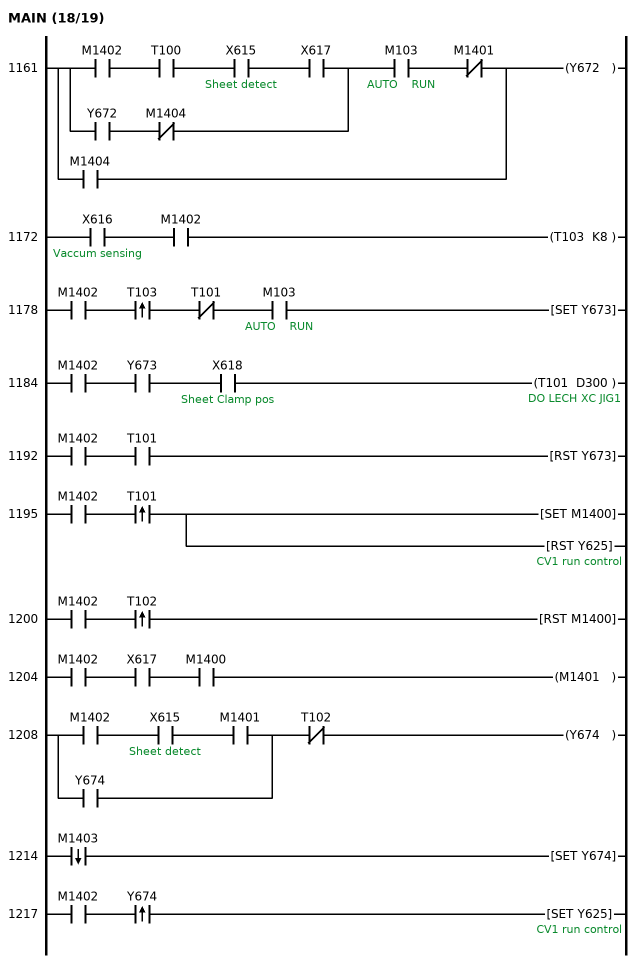
[picture p24: ladder of MAIN, rungs at steps 1161 to 1217]
1161  LD      M1402
      AND     T100
      AND     X615  ; Sheet detect
      AND     X617
      LD      Y672
      ANI     M1404
      ORB
      AND     M103  ; AUTO    RUN
      ANI     M1401
      OR      M1404
      OUT     Y672
1172  LD      X616  ; Vaccum sensing
      AND     M1402
      OUT     T103 K8
1178  LD      M1402
      ANDP    T103
      ANI     T101
      AND     M103  ; AUTO    RUN
      SET     Y673
1184  LD      M1402
      AND     Y673
      AND     X618  ; Sheet Clamp pos
      OUT     T101 D300  ; DO LECH XC JIG1
1192  LD      M1402
      AND     T101
      RST     Y673
1195  LD      M1402
      ANDP    T101
      SET     M1400
      RST     Y625  ; CV1 run control
1200  LD      M1402
      ANDP    T102
      RST     M1400
1204  LD      M1402
      AND     X617
      AND     M1400
      OUT     M1401
1208  LD      M1402
      AND     X615  ; Sheet detect
      AND     M1401
      OR      Y674
      ANI     T102
      OUT     Y674
1214  LDF     M1403
      SET     Y674
1217  LD      M1402
      ANDP    Y674
      SET     Y625  ; CV1 run control
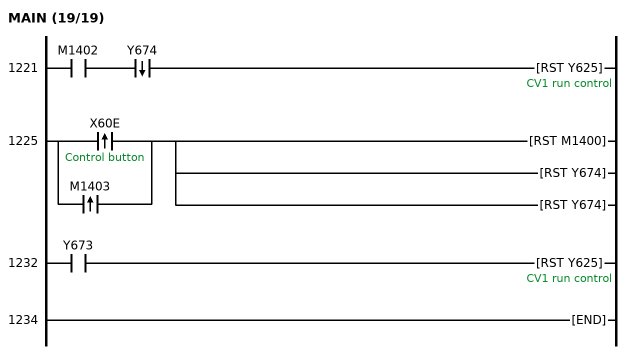
1221  LD      M1402
      ANDF    Y674
      RST     Y625  ; CV1 run control
1225  LDP     X60E  ; Control button
      ORP     M1403
      RST     M1400
      RST     Y674
      RST     Y674
1232  LD      Y673
      RST     Y625  ; CV1 run control
1234  END
END_PROGRAM

PROGRAM MONITOR
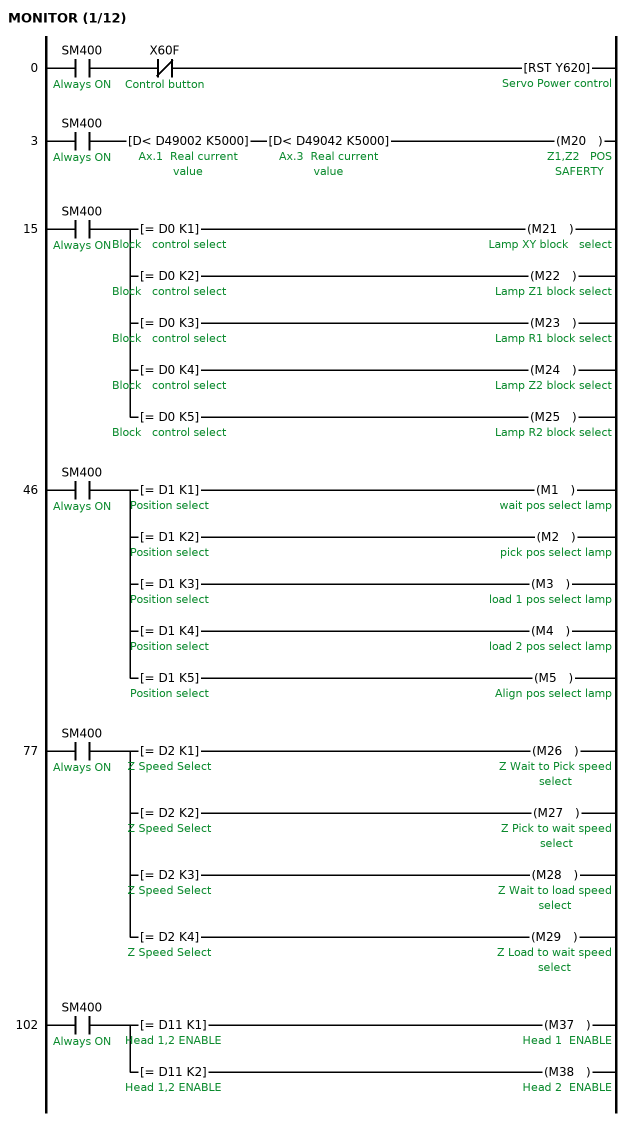
0     LD      SM400  ; Always ON
      ANI     X60F  ; Control button
      RST     Y620  ; Servo Power control
3     LD      SM400  ; Always ON
      ANDD<   D49002 K5000  ; Ax.1  Real current value
      ANDD<   D49042 K5000  ; Ax.3  Real current value
      OUT     M20  ; Z1,Z2   POS     SAFERTY
15    LD      SM400  ; Always ON
      MPS
      AND=    D0 K1  ; Block   control select
      OUT     M21  ; Lamp XY block   select
      MRD
      AND=    D0 K2  ; Block   control select
      OUT     M22  ; Lamp Z1 block select
      MRD
      AND=    D0 K3  ; Block   control select
      OUT     M23  ; Lamp R1 block select
      MRD
      AND=    D0 K4  ; Block   control select
      OUT     M24  ; Lamp Z2 block select
      MPP
      AND=    D0 K5  ; Block   control select
      OUT     M25  ; Lamp R2 block select
46    LD      SM400  ; Always ON
      MPS
      AND=    D1 K1  ; Position select
      OUT     M1  ; wait pos select lamp
      MRD
      AND=    D1 K2  ; Position select
      OUT     M2  ; pick pos select lamp
      MRD
      AND=    D1 K3  ; Position select
      OUT     M3  ; load 1 pos select lamp
      MRD
      AND=    D1 K4  ; Position select
      OUT     M4  ; load 2 pos select lamp
      MPP
      AND=    D1 K5  ; Position select
      OUT     M5  ; Align pos select lamp
77    LD      SM400  ; Always ON
      MPS
      AND=    D2 K1  ; Z Speed Select
      OUT     M26  ; Z Wait to Pick speed select
      MRD
      AND=    D2 K2  ; Z Speed Select
      OUT     M27  ; Z Pick to wait speed select
      MRD
      AND=    D2 K3  ; Z Speed Select
      OUT     M28  ; Z Wait to load speed select
      MPP
      AND=    D2 K4  ; Z Speed Select
      OUT     M29  ; Z Load to wait speed select
102   LD      SM400  ; Always ON
      MPS
      AND=    D11 K1  ; Head 1,2 ENABLE
      OUT     M37  ; Head 1  ENABLE
      MPP
      AND=    D11 K2  ; Head 1,2 ENABLE
      OUT     M38  ; Head 2  ENABLE
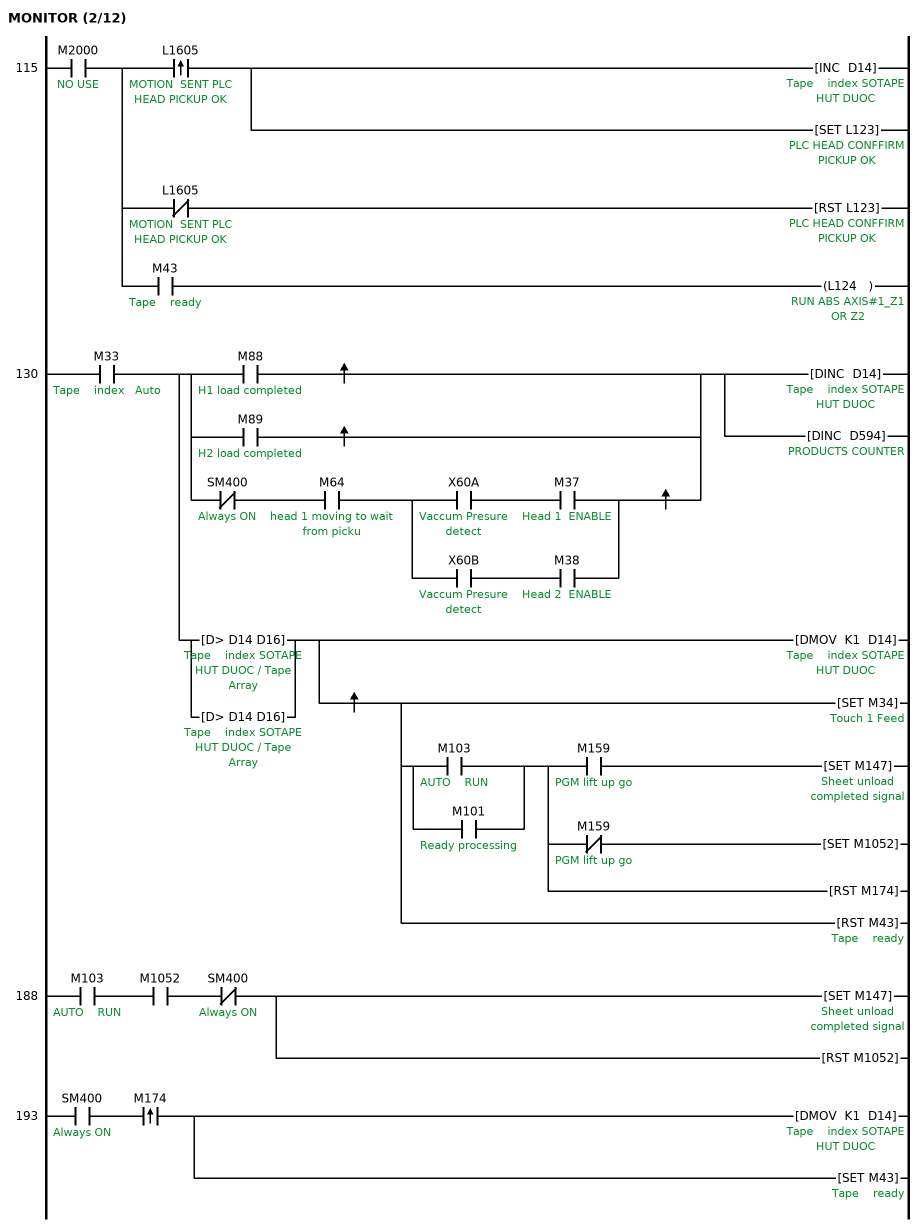
115   LD      M2000  ; NO USE
      MPS
      ANDP    L1605  ; MOTION  SENT PLC HEAD PICKUP OK
      INC     D14  ; Tape    index SOTAPE HUT DUOC
      SET     L123  ; PLC HEAD CONFFIRM PICKUP OK
      MRD
      ANI     L1605  ; MOTION  SENT PLC HEAD PICKUP OK
      RST     L123  ; PLC HEAD CONFFIRM PICKUP OK
      MPP
      AND     M43  ; Tape    ready
      OUT     L124  ; RUN ABS AXIS#1_Z1 OR Z2
130   LD      M33  ; Tape    index   Auto
      MPS
      LD      M88  ; H1 load completed
      MEP
      LD      M89  ; H2 load completed
      MEP
      ORB
      LDI     SM400  ; Always ON
      AND     M64  ; head 1 moving to wait from picku
      LD      X60A  ; Vaccum Presure detect
      AND     M37  ; Head 1  ENABLE
      LD      X60B  ; Vaccum Presure detect
      AND     M38  ; Head 2  ENABLE
      ORB
      ANB
      MEP
      ORB
      ANB
      DINC    D14
      DINC    D594  ; PRODUCTS COUNTER
      MPP
      LDD>    D14 D16  ; Tape    index SOTAPE HUT DUOC / Tape Array
      ORD>    D14 D16  ; Tape    index SOTAPE HUT DUOC / Tape Array
      ANB
      DMOV    K1 D14
      MEP
      SET     M34  ; Touch 1 Feed
      MPS
      LD      M103  ; AUTO    RUN
      OR      M101  ; Ready processing
      ANB
      MPS
      AND     M159  ; PGM lift up go
      SET     M147  ; Sheet unload completed signal
      MRD
      ANI     M159  ; PGM lift up go
      SET     M1052
      MPP
      RST     M174
      MPP
      RST     M43  ; Tape    ready
188   LD      M103  ; AUTO    RUN
      AND     M1052
      ANI     SM400  ; Always ON
      SET     M147  ; Sheet unload completed signal
      RST     M1052
193   LD      SM400  ; Always ON
      ANDP    M174
      DMOV    K1 D14
      SET     M43  ; Tape    ready
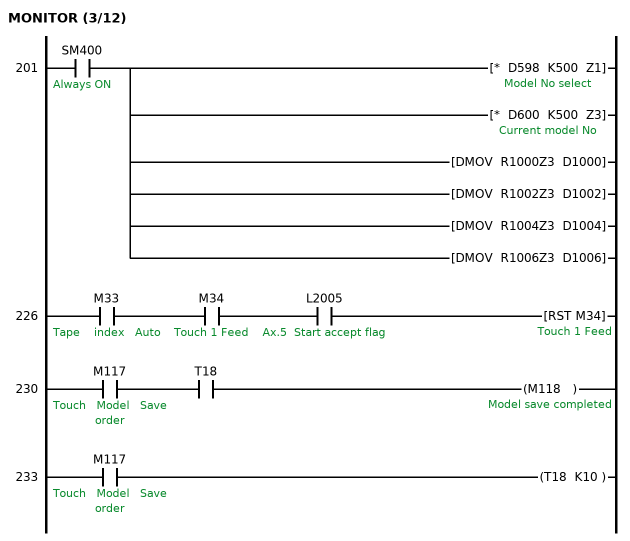
201   LD      SM400  ; Always ON
      *       D598 K500 Z1  ; Model No select
      *       D600 K500 Z3  ; Current model No
      DMOV    R1000Z3 D1000
      DMOV    R1002Z3 D1002
      DMOV    R1004Z3 D1004
      DMOV    R1006Z3 D1006
226   LD      M33  ; Tape    index   Auto
      AND     M34  ; Touch 1 Feed
      AND     L2005  ; Ax.5  Start accept flag
      RST     M34  ; Touch 1 Feed
230   LD      M117  ; Touch   Model   Save    order
      AND     T18
      OUT     M118  ; Model save completed
233   LD      M117  ; Touch   Model   Save    order
      OUT     T18 K10
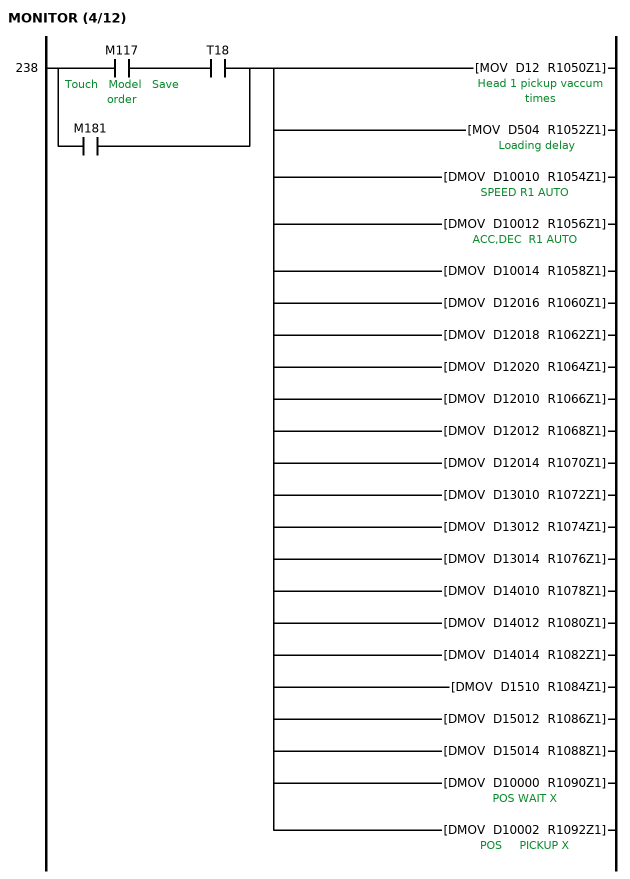
238   LD      M117  ; Touch   Model   Save    order
      AND     T18
      OR      M181
      MOV     D12 R1050Z1  ; Head 1 pickup vaccum times
      MOV     D504 R1052Z1  ; Loading delay
      DMOV    D10010 R1054Z1  ; SPEED R1 AUTO
      DMOV    D10012 R1056Z1  ; ACC,DEC  R1 AUTO
      DMOV    D10014 R1058Z1
      DMOV    D12016 R1060Z1
      DMOV    D12018 R1062Z1
      DMOV    D12020 R1064Z1
      DMOV    D12010 R1066Z1
      DMOV    D12012 R1068Z1
      DMOV    D12014 R1070Z1
      DMOV    D13010 R1072Z1
      DMOV    D13012 R1074Z1
      DMOV    D13014 R1076Z1
      DMOV    D14010 R1078Z1
      DMOV    D14012 R1080Z1
      DMOV    D14014 R1082Z1
      DMOV    D1510 R1084Z1
      DMOV    D15012 R1086Z1
      DMOV    D15014 R1088Z1
      DMOV    D10000 R1090Z1  ; POS WAIT X
      DMOV    D10002 R1092Z1  ; POS     PICKUP X
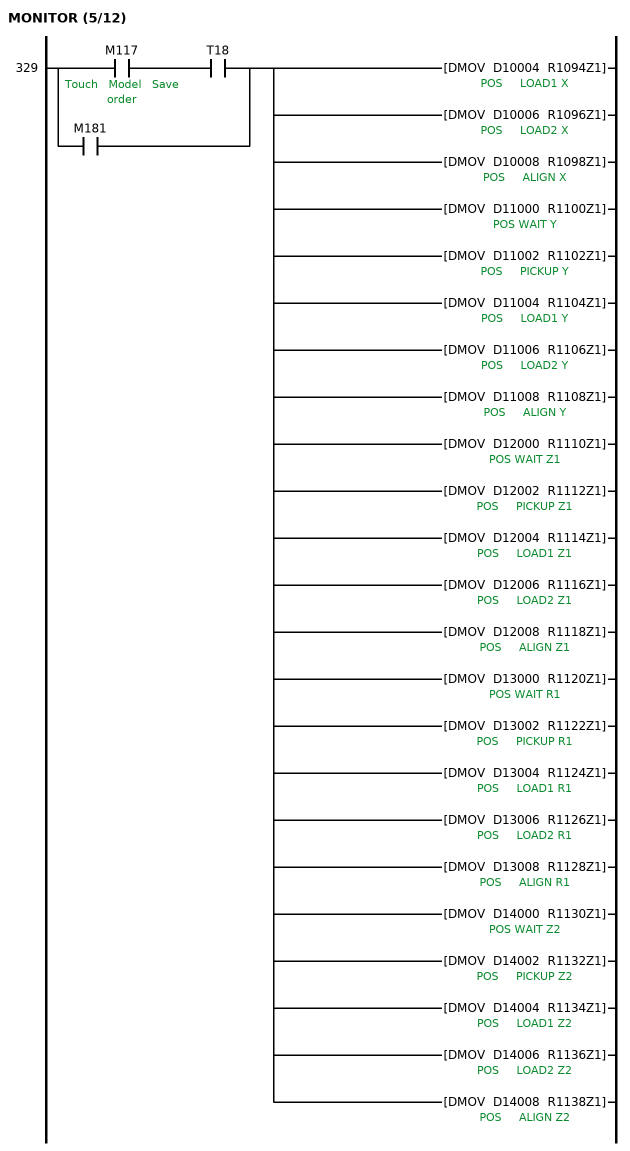
329   LD      M117  ; Touch   Model   Save    order
      AND     T18
      OR      M181
      DMOV    D10004 R1094Z1  ; POS     LOAD1 X
      DMOV    D10006 R1096Z1  ; POS     LOAD2 X
      DMOV    D10008 R1098Z1  ; POS     ALIGN X
      DMOV    D11000 R1100Z1  ; POS WAIT Y
      DMOV    D11002 R1102Z1  ; POS     PICKUP Y
      DMOV    D11004 R1104Z1  ; POS     LOAD1 Y
      DMOV    D11006 R1106Z1  ; POS     LOAD2 Y
      DMOV    D11008 R1108Z1  ; POS     ALIGN Y
      DMOV    D12000 R1110Z1  ; POS WAIT Z1
      DMOV    D12002 R1112Z1  ; POS     PICKUP Z1
      DMOV    D12004 R1114Z1  ; POS     LOAD1 Z1
      DMOV    D12006 R1116Z1  ; POS     LOAD2 Z1
      DMOV    D12008 R1118Z1  ; POS     ALIGN Z1
      DMOV    D13000 R1120Z1  ; POS WAIT R1
      DMOV    D13002 R1122Z1  ; POS     PICKUP R1
      DMOV    D13004 R1124Z1  ; POS     LOAD1 R1
      DMOV    D13006 R1126Z1  ; POS     LOAD2 R1
      DMOV    D13008 R1128Z1  ; POS     ALIGN R1
      DMOV    D14000 R1130Z1  ; POS WAIT Z2
      DMOV    D14002 R1132Z1  ; POS     PICKUP Z2
      DMOV    D14004 R1134Z1  ; POS     LOAD1 Z2
      DMOV    D14006 R1136Z1  ; POS     LOAD2 Z2
      DMOV    D14008 R1138Z1  ; POS     ALIGN Z2
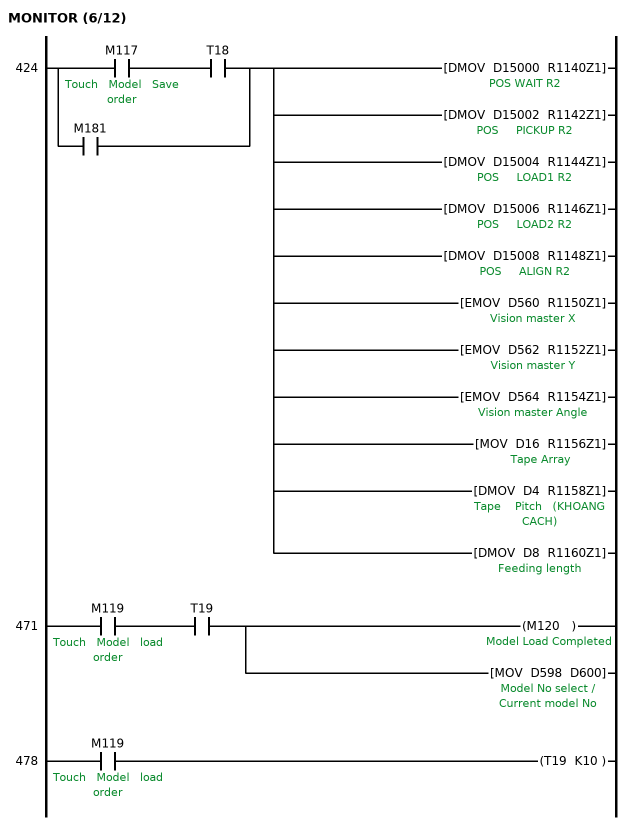
424   LD      M117  ; Touch   Model   Save    order
      AND     T18
      OR      M181
      DMOV    D15000 R1140Z1  ; POS WAIT R2
      DMOV    D15002 R1142Z1  ; POS     PICKUP R2
      DMOV    D15004 R1144Z1  ; POS     LOAD1 R2
      DMOV    D15006 R1146Z1  ; POS     LOAD2 R2
      DMOV    D15008 R1148Z1  ; POS     ALIGN R2
      EMOV    D560 R1150Z1  ; Vision master X
      EMOV    D562 R1152Z1  ; Vision master Y
      EMOV    D564 R1154Z1  ; Vision master Angle
      MOV     D16 R1156Z1
      DMOV    D4 R1158Z1  ; Tape    Pitch   (KHOANG  CACH)
      DMOV    D8 R1160Z1  ; Feeding length
471   LD      M119  ; Touch   Model   load    order
      AND     T19
      OUT     M120  ; Model Load Completed
      MOV     D598 D600
478   LD      M119  ; Touch   Model   load    order
      OUT     T19 K10
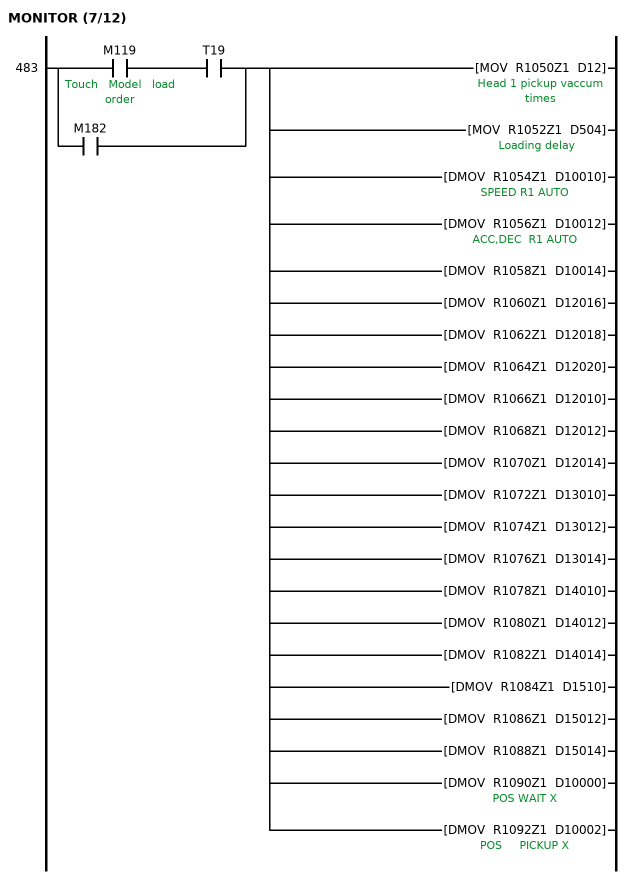
483   LD      M119  ; Touch   Model   load    order
      AND     T19
      OR      M182
      MOV     R1050Z1 D12
      MOV     R1052Z1 D504
      DMOV    R1054Z1 D10010
      DMOV    R1056Z1 D10012
      DMOV    R1058Z1 D10014
      DMOV    R1060Z1 D12016
      DMOV    R1062Z1 D12018
      DMOV    R1064Z1 D12020
      DMOV    R1066Z1 D12010
      DMOV    R1068Z1 D12012
      DMOV    R1070Z1 D12014
      DMOV    R1072Z1 D13010
      DMOV    R1074Z1 D13012
      DMOV    R1076Z1 D13014
      DMOV    R1078Z1 D14010
      DMOV    R1080Z1 D14012
      DMOV    R1082Z1 D14014
      DMOV    R1084Z1 D1510
      DMOV    R1086Z1 D15012
      DMOV    R1088Z1 D15014
      DMOV    R1090Z1 D10000
      DMOV    R1092Z1 D10002
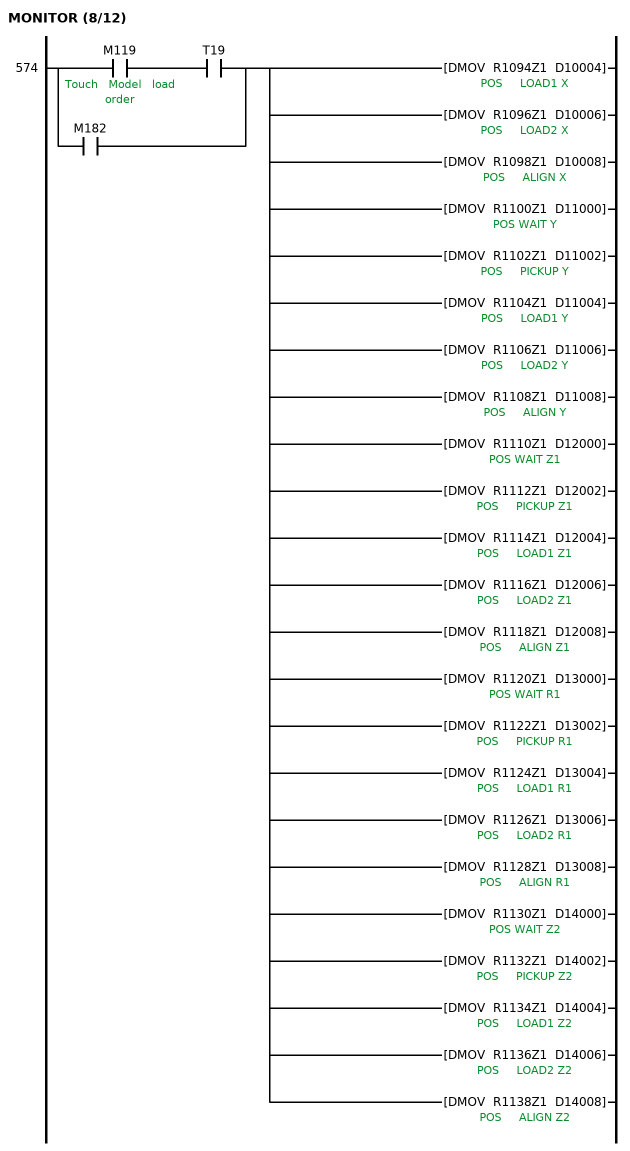
574   LD      M119  ; Touch   Model   load    order
      AND     T19
      OR      M182
      DMOV    R1094Z1 D10004
      DMOV    R1096Z1 D10006
      DMOV    R1098Z1 D10008
      DMOV    R1100Z1 D11000
      DMOV    R1102Z1 D11002
      DMOV    R1104Z1 D11004
      DMOV    R1106Z1 D11006
      DMOV    R1108Z1 D11008
      DMOV    R1110Z1 D12000
      DMOV    R1112Z1 D12002
      DMOV    R1114Z1 D12004
      DMOV    R1116Z1 D12006
      DMOV    R1118Z1 D12008
      DMOV    R1120Z1 D13000
      DMOV    R1122Z1 D13002
      DMOV    R1124Z1 D13004
      DMOV    R1126Z1 D13006
      DMOV    R1128Z1 D13008
      DMOV    R1130Z1 D14000
      DMOV    R1132Z1 D14002
      DMOV    R1134Z1 D14004
      DMOV    R1136Z1 D14006
      DMOV    R1138Z1 D14008
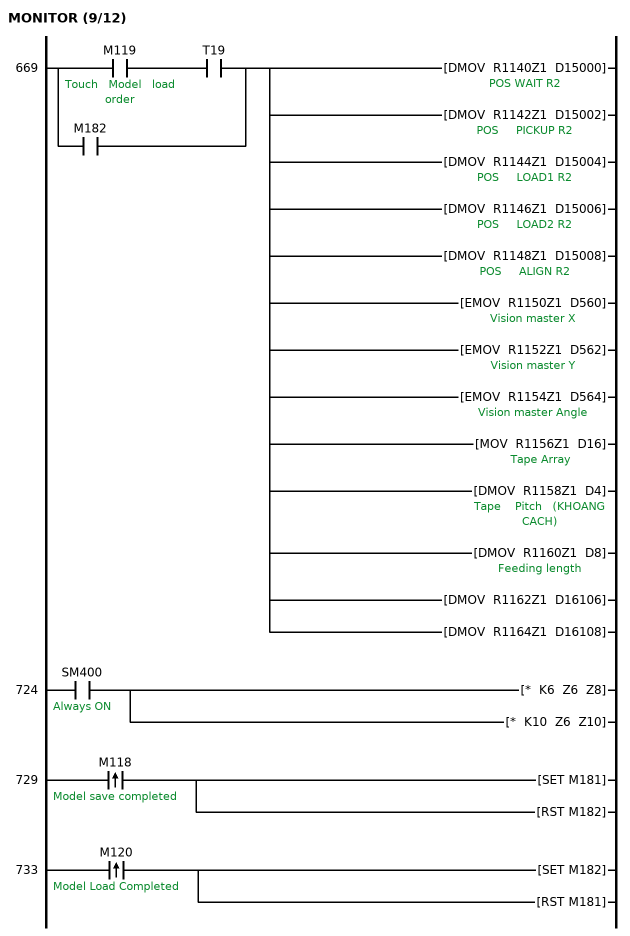
669   LD      M119  ; Touch   Model   load    order
      AND     T19
      OR      M182
      DMOV    R1140Z1 D15000
      DMOV    R1142Z1 D15002
      DMOV    R1144Z1 D15004
      DMOV    R1146Z1 D15006
      DMOV    R1148Z1 D15008
      EMOV    R1150Z1 D560
      EMOV    R1152Z1 D562
      EMOV    R1154Z1 D564
      MOV     R1156Z1 D16
      DMOV    R1158Z1 D4
      DMOV    R1160Z1 D8
      DMOV    R1162Z1 D16106
      DMOV    R1164Z1 D16108
724   LD      SM400  ; Always ON
      *       K6 Z6 Z8
      *       K10 Z6 Z10
729   LDP     M118  ; Model save completed
      SET     M181
      RST     M182
733   LDP     M120  ; Model Load Completed
      SET     M182
      RST     M181
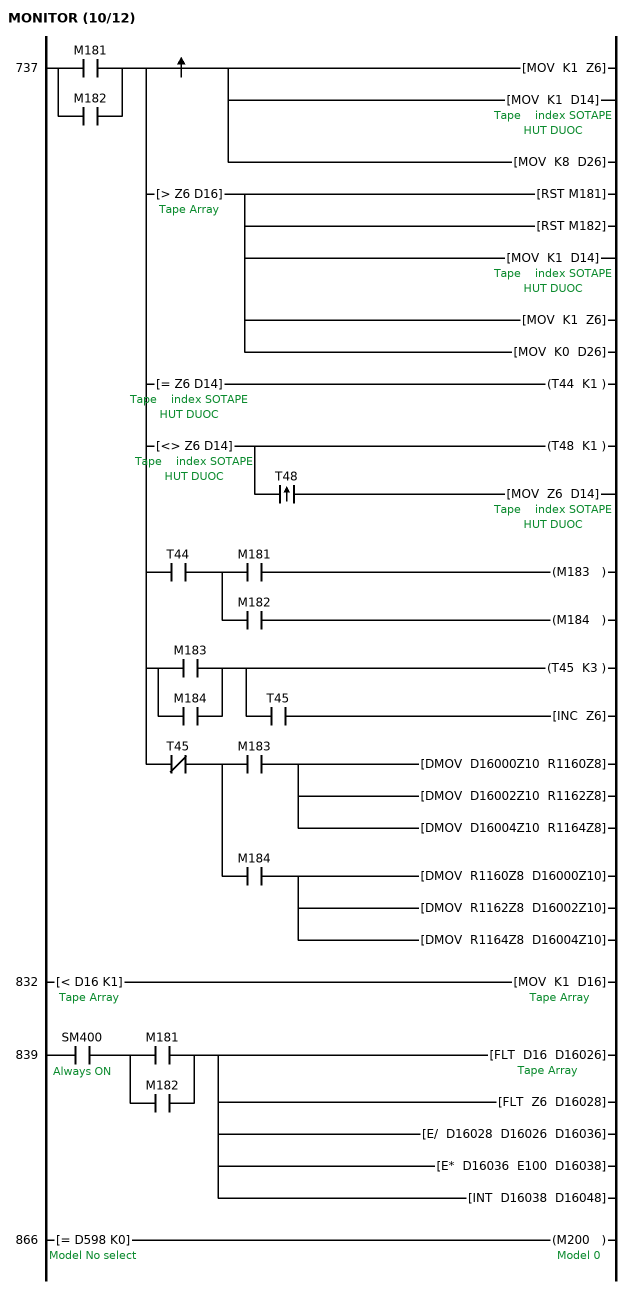
737   LD      M181
      OR      M182
      MPS
      MEP
      MOV     K1 Z6
      MOV     K1 D14
      MOV     K8 D26
      MRD
      AND>    Z6 D16  ; Tape Array
      RST     M181
      RST     M182
      MOV     K1 D14
      MOV     K1 Z6
      MOV     K0 D26
      MRD
      AND=    Z6 D14  ; Tape    index SOTAPE HUT DUOC
      OUT     T44 K1
      MRD
      AND<>   Z6 D14  ; Tape    index SOTAPE HUT DUOC
      OUT     T48 K1
      ANDP    T48
      MOV     Z6 D14
      MRD
      AND     T44
      MPS
      AND     M181
      OUT     M183
      MPP
      AND     M182
      OUT     M184
      MRD
      LD      M183
      OR      M184
      ANB
      OUT     T45 K3
      AND     T45
      INC     Z6
      MPP
      ANI     T45
      MPS
      AND     M183
      DMOV    D16000Z10 R1160Z8
      DMOV    D16002Z10 R1162Z8
      DMOV    D16004Z10 R1164Z8
      MPP
      AND     M184
      DMOV    R1160Z8 D16000Z10
      DMOV    R1162Z8 D16002Z10
      DMOV    R1164Z8 D16004Z10
832   LD<     D16 K1  ; Tape Array
      MOV     K1 D16
839   LD      SM400  ; Always ON
      LD      M181
      OR      M182
      ANB
      FLT     D16 D16026
      FLT     Z6 D16028
      E/      D16028 D16026 D16036
      E*      D16036 E100 D16038
      INT     D16038 D16048
866   LD=     D598 K0  ; Model No select
      OUT     M200  ; Model 0
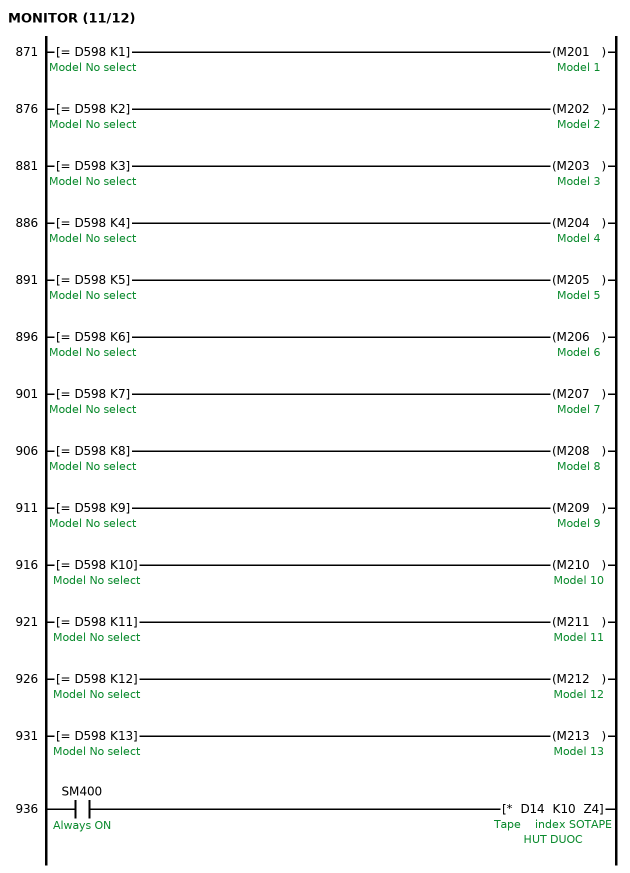
871   LD=     D598 K1  ; Model No select
      OUT     M201  ; Model 1
876   LD=     D598 K2  ; Model No select
      OUT     M202  ; Model 2
881   LD=     D598 K3  ; Model No select
      OUT     M203  ; Model 3
886   LD=     D598 K4  ; Model No select
      OUT     M204  ; Model 4
891   LD=     D598 K5  ; Model No select
      OUT     M205  ; Model 5
896   LD=     D598 K6  ; Model No select
      OUT     M206  ; Model 6
901   LD=     D598 K7  ; Model No select
      OUT     M207  ; Model 7
906   LD=     D598 K8  ; Model No select
      OUT     M208  ; Model 8
911   LD=     D598 K9  ; Model No select
      OUT     M209  ; Model 9
916   LD=     D598 K10  ; Model No select
      OUT     M210  ; Model 10
921   LD=     D598 K11  ; Model No select
      OUT     M211  ; Model 11
926   LD=     D598 K12  ; Model No select
      OUT     M212  ; Model 12
931   LD=     D598 K13  ; Model No select
      OUT     M213  ; Model 13
936   LD      SM400  ; Always ON
      *       D14 K10 Z4
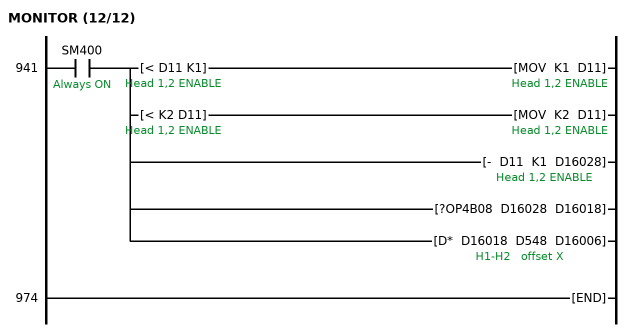
941   LD      SM400  ; Always ON
      MPS
      AND<    D11 K1  ; Head 1,2 ENABLE
      MOV     K1 D11
      MRD
      AND<    K2 D11  ; Head 1,2 ENABLE
      MOV     K2 D11
      MPP
      -       D11 K1 D16028
      ?OP4B08 D16028 D16018
      D*      D16018 D548 D16006  ; H1-H2   offset X
974   END
END_PROGRAM

PROGRAM MOTION
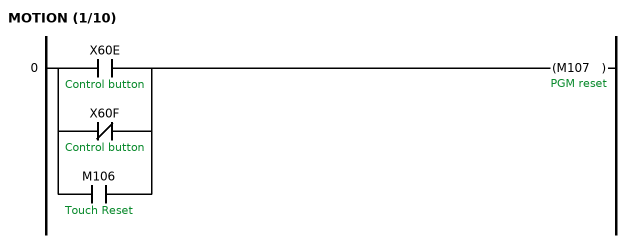
0     LD      X60E  ; Control button
      ORI     X60F  ; Control button
      OR      M106  ; Touch Reset
      OUT     M107  ; PGM reset
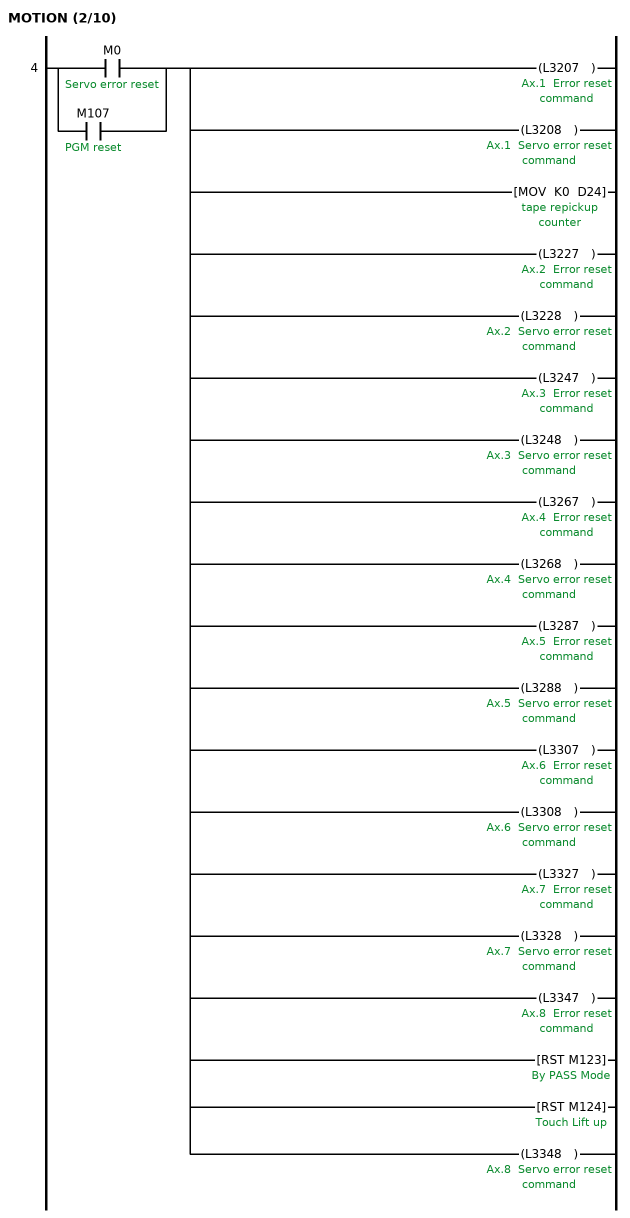
4     LD      M0  ; Servo error reset
      OR      M107  ; PGM reset
      OUT     L3207  ; Ax.1  Error reset command
      OUT     L3208  ; Ax.1  Servo error reset command
      MOV     K0 D24  ; tape repickup counter
      OUT     L3227  ; Ax.2  Error reset command
      OUT     L3228  ; Ax.2  Servo error reset command
      OUT     L3247  ; Ax.3  Error reset command
      OUT     L3248  ; Ax.3  Servo error reset command
      OUT     L3267  ; Ax.4  Error reset command
      OUT     L3268  ; Ax.4  Servo error reset command
      OUT     L3287  ; Ax.5  Error reset command
      OUT     L3288  ; Ax.5  Servo error reset command
      OUT     L3307  ; Ax.6  Error reset command
      OUT     L3308  ; Ax.6  Servo error reset command
      OUT     L3327  ; Ax.7  Error reset command
      OUT     L3328  ; Ax.7  Servo error reset command
      OUT     L3347  ; Ax.8  Error reset command
      RST     M123  ; By PASS Mode
      RST     M124  ; Touch Lift up
      OUT     L3348  ; Ax.8  Servo error reset command
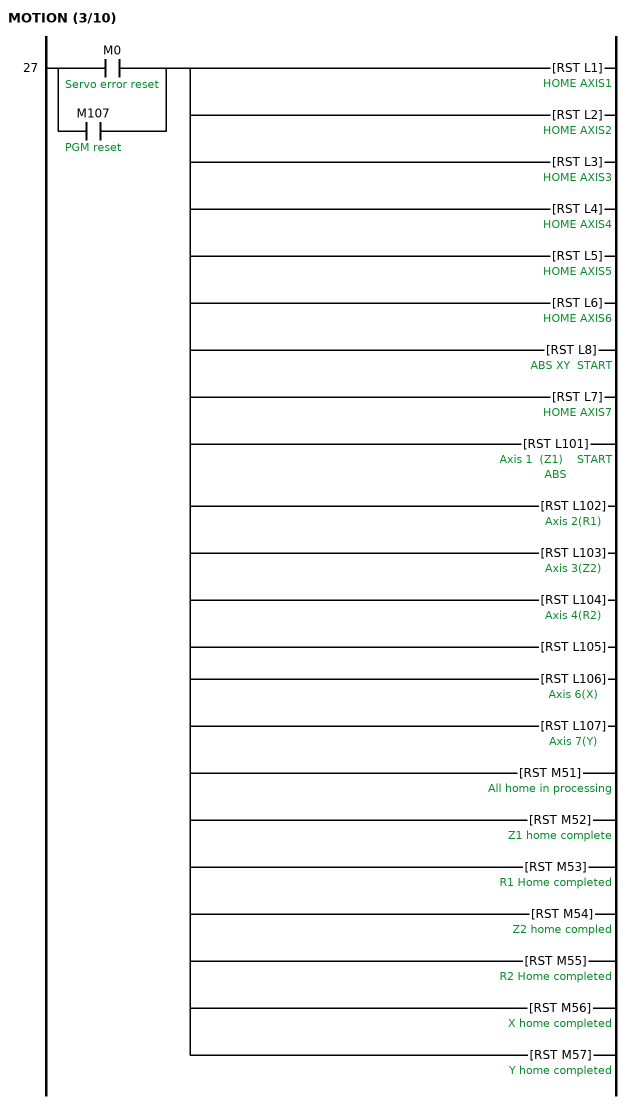
27    LD      M0  ; Servo error reset
      OR      M107  ; PGM reset
      RST     L1  ; HOME AXIS1
      RST     L2  ; HOME AXIS2
      RST     L3  ; HOME AXIS3
      RST     L4  ; HOME AXIS4
      RST     L5  ; HOME AXIS5
      RST     L6  ; HOME AXIS6
      RST     L8  ; ABS XY  START
      RST     L7  ; HOME AXIS7
      RST     L101  ; Axis 1  (Z1)    START   ABS
      RST     L102  ; Axis 2(R1)
      RST     L103  ; Axis 3(Z2)
      RST     L104  ; Axis 4(R2)
      RST     L105
      RST     L106  ; Axis 6(X)
      RST     L107  ; Axis 7(Y)
      RST     M51  ; All home in processing
      RST     M52  ; Z1 home complete
      RST     M53  ; R1 Home completed
      RST     M54  ; Z2 home compled
      RST     M55  ; R2 Home completed
      RST     M56  ; X home completed
      RST     M57  ; Y home completed
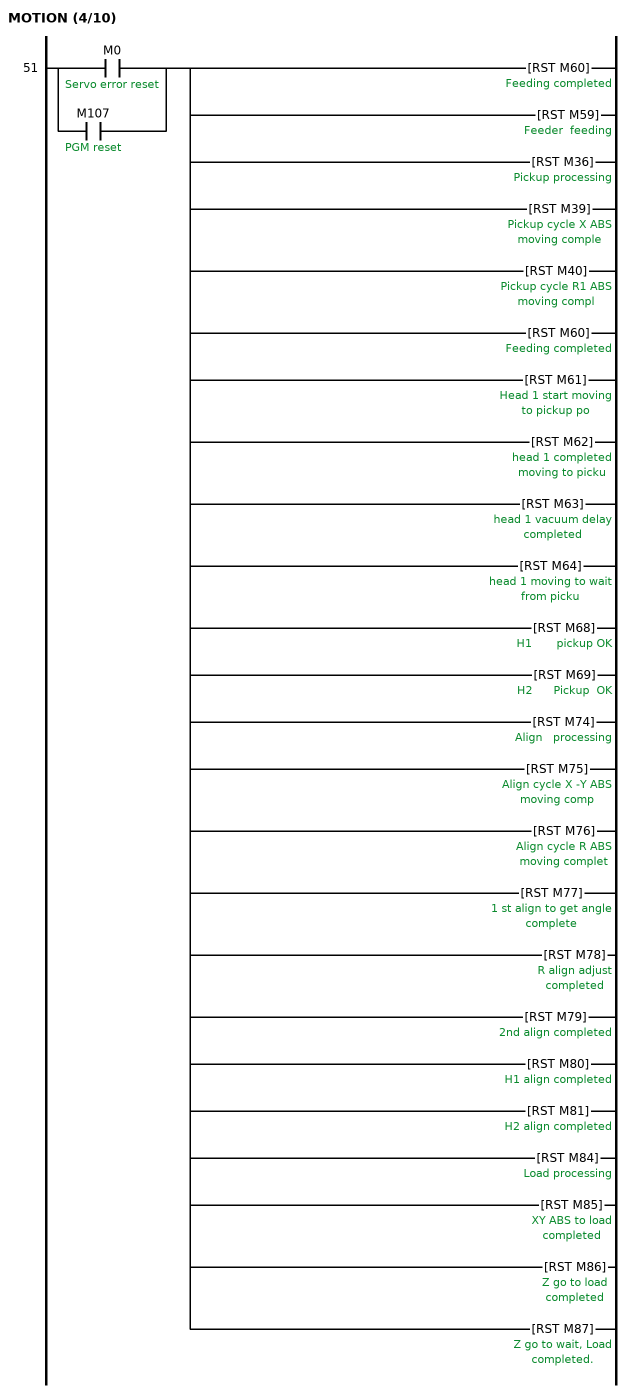
51    LD      M0  ; Servo error reset
      OR      M107  ; PGM reset
      RST     M60  ; Feeding completed
      RST     M59  ; Feeder  feeding
      RST     M36  ; Pickup processing
      RST     M39  ; Pickup cycle X ABS moving comple
      RST     M40  ; Pickup cycle R1 ABS moving compl
      RST     M60  ; Feeding completed
      RST     M61  ; Head 1 start moving to pickup po
      RST     M62  ; head 1 completed moving to picku
      RST     M63  ; head 1 vacuum delay completed
      RST     M64  ; head 1 moving to wait from picku
      RST     M68  ; H1       pickup OK
      RST     M69  ; H2      Pickup  OK
      RST     M74  ; Align   processing
      RST     M75  ; Align cycle X -Y ABS moving comp
      RST     M76  ; Align cycle R ABS moving complet
      RST     M77  ; 1 st align to get angle complete
      RST     M78  ; R align adjust completed
      RST     M79  ; 2nd align completed
      RST     M80  ; H1 align completed
      RST     M81  ; H2 align completed
      RST     M84  ; Load processing
      RST     M85  ; XY ABS to load completed
      RST     M86  ; Z go to load completed
      RST     M87  ; Z go to wait, Load completed.
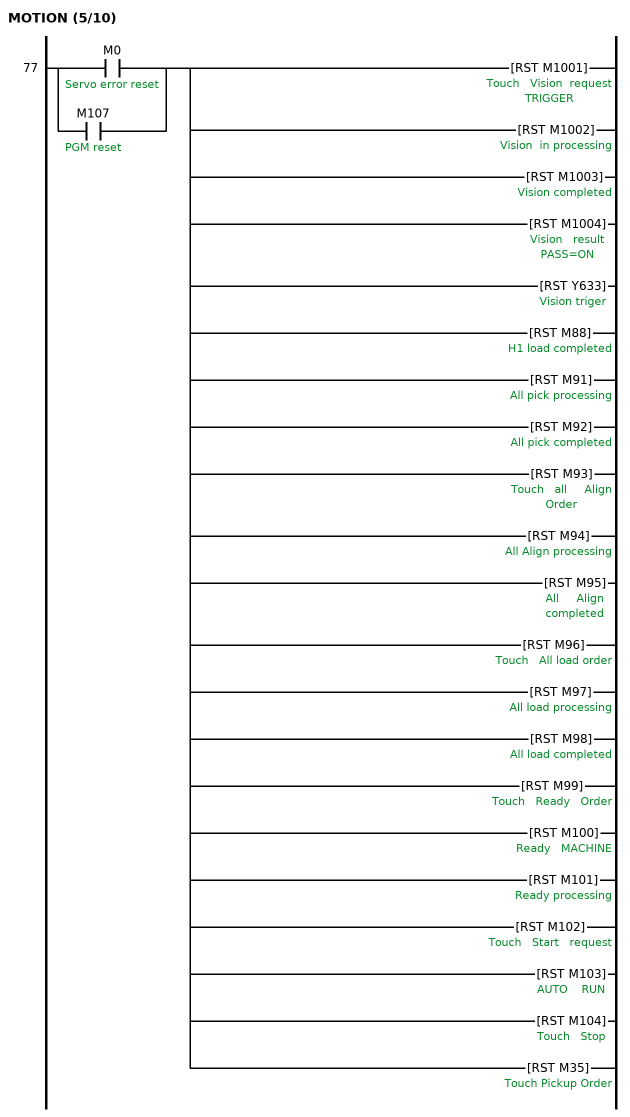
77    LD      M0  ; Servo error reset
      OR      M107  ; PGM reset
      RST     M1001  ; Touch   Vision  request TRIGGER
      RST     M1002  ; Vision  in processing
      RST     M1003  ; Vision completed
      RST     M1004  ; Vision   result PASS=ON
      RST     Y633  ; Vision triger
      RST     M88  ; H1 load completed
      RST     M91  ; All pick processing
      RST     M92  ; All pick completed
      RST     M93  ; Touch   all     Align   Order
      RST     M94  ; All Align processing
      RST     M95  ; All     Align   completed
      RST     M96  ; Touch   All load order
      RST     M97  ; All load processing
      RST     M98  ; All load completed
      RST     M99  ; Touch   Ready   Order
      RST     M100  ; Ready   MACHINE
      RST     M101  ; Ready processing
      RST     M102  ; Touch   Start   request
      RST     M103  ; AUTO    RUN
      RST     M104  ; Touch   Stop
      RST     M35  ; Touch Pickup Order
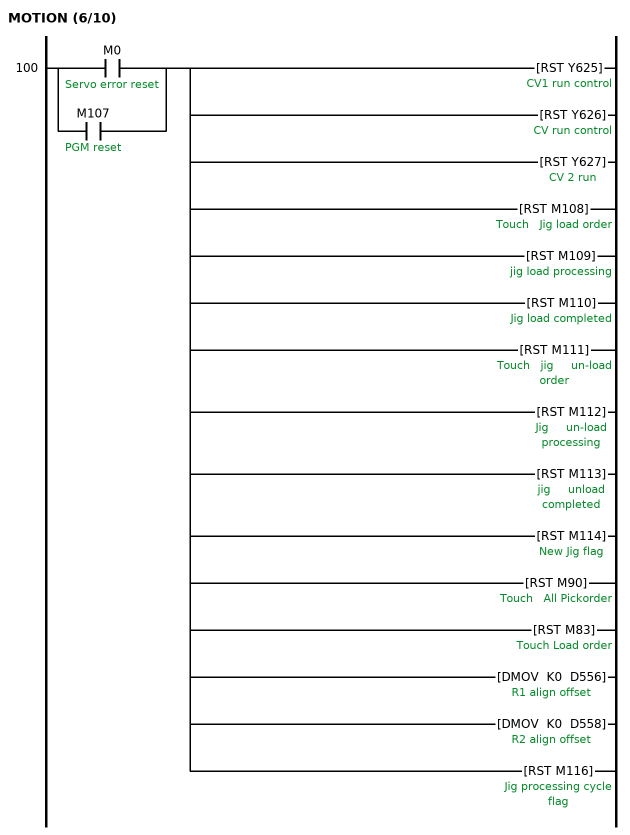
100   LD      M0  ; Servo error reset
      OR      M107  ; PGM reset
      RST     Y625  ; CV1 run control
      RST     Y626  ; CV run control
      RST     Y627  ; CV 2 run
      RST     M108  ; Touch   Jig load order
      RST     M109  ; jig load processing
      RST     M110  ; Jig load completed
      RST     M111  ; Touch   jig     un-load order
      RST     M112  ; Jig     un-load processing
      RST     M113  ; jig     unload  completed
      RST     M114  ; New Jig flag
      RST     M90  ; Touch   All Pickorder
      RST     M83  ; Touch Load order
      DMOV    K0 D556  ; R1 align offset
      DMOV    K0 D558  ; R2 align offset
      RST     M116  ; Jig processing cycle flag
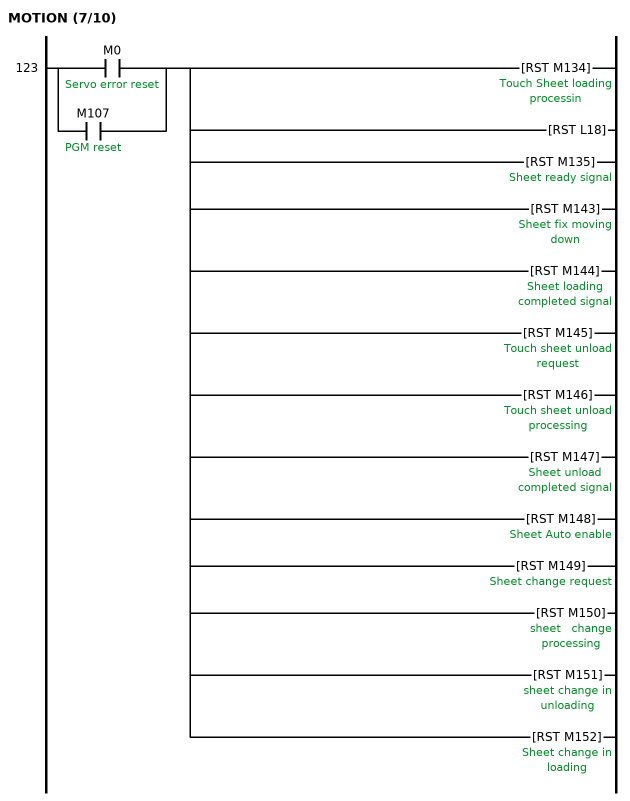
123   LD      M0  ; Servo error reset
      OR      M107  ; PGM reset
      RST     M134  ; Touch Sheet loading processin
      RST     L18
      RST     M135  ; Sheet ready signal
      RST     M143  ; Sheet fix moving down
      RST     M144  ; Sheet loading completed signal
      RST     M145  ; Touch sheet unload request
      RST     M146  ; Touch sheet unload processing
      RST     M147  ; Sheet unload completed signal
      RST     M148  ; Sheet Auto enable
      RST     M149  ; Sheet change request
      RST     M150  ; sheet   change  processing
      RST     M151  ; sheet change in unloading
      RST     M152  ; Sheet change in loading
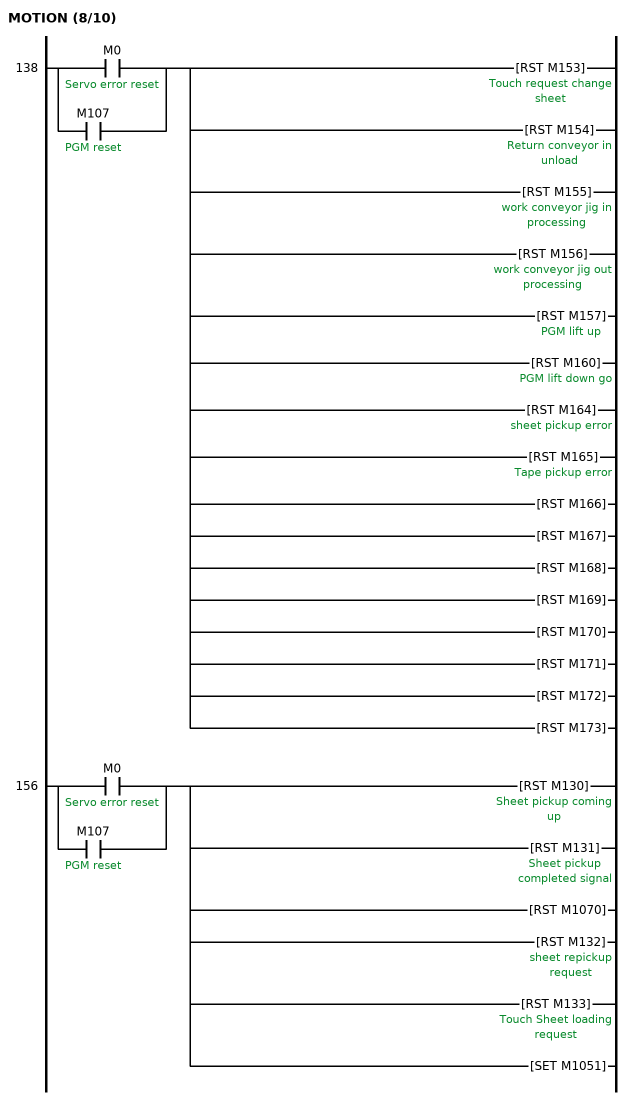
138   LD      M0  ; Servo error reset
      OR      M107  ; PGM reset
      RST     M153  ; Touch request change sheet
      RST     M154  ; Return conveyor in unload
      RST     M155  ; work conveyor jig in processing
      RST     M156  ; work conveyor jig out processing
      RST     M157  ; PGM lift up
      RST     M160  ; PGM lift down go
      RST     M164  ; sheet pickup error
      RST     M165  ; Tape pickup error
      RST     M166
      RST     M167
      RST     M168
      RST     M169
      RST     M170
      RST     M171
      RST     M172
      RST     M173
156   LD      M0  ; Servo error reset
      OR      M107  ; PGM reset
      RST     M130  ; Sheet pickup coming up
      RST     M131  ; Sheet pickup completed signal
      RST     M1070
      RST     M132  ; sheet repickup request
      RST     M133  ; Touch Sheet loading request
      SET     M1051
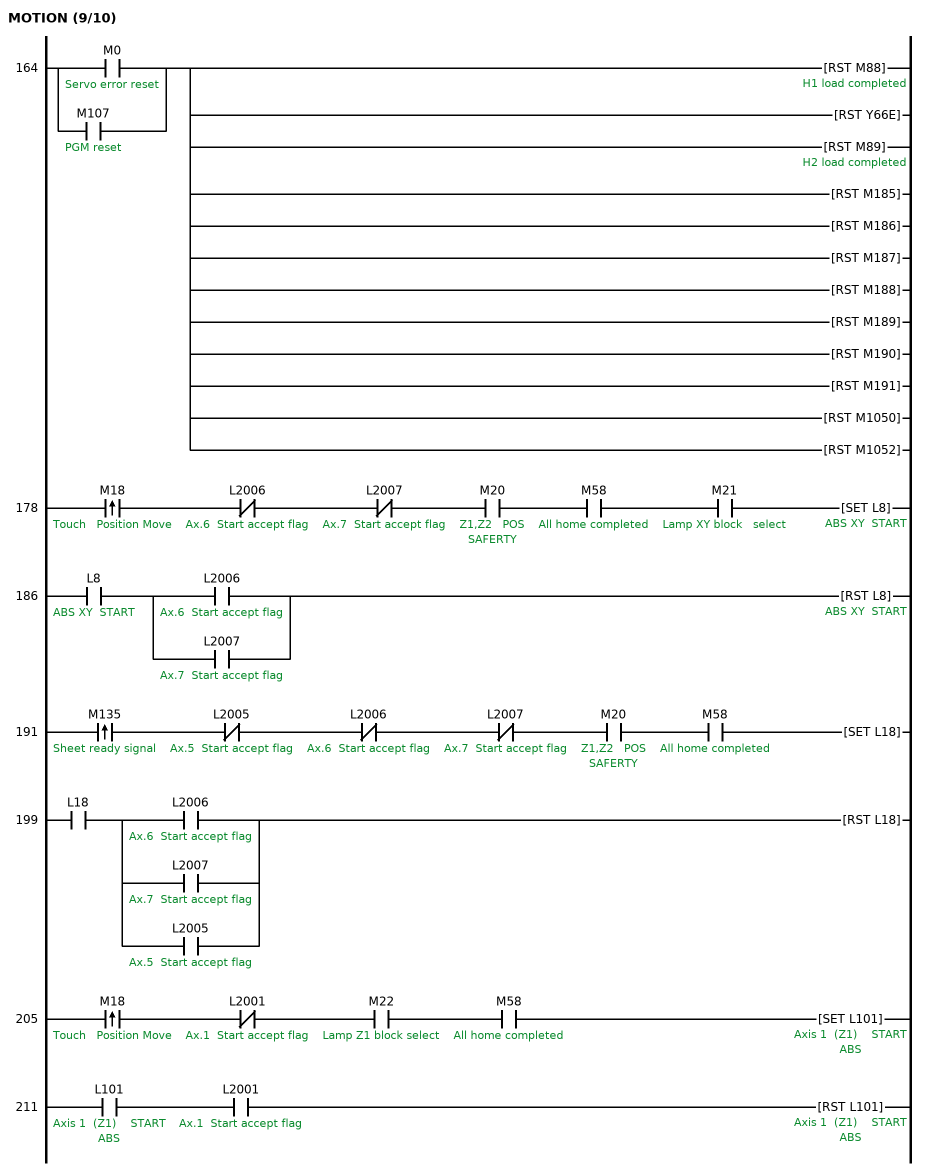
164   LD      M0  ; Servo error reset
      OR      M107  ; PGM reset
      RST     M88  ; H1 load completed
      RST     Y66E
      RST     M89  ; H2 load completed
      RST     M185
      RST     M186
      RST     M187
      RST     M188
      RST     M189
      RST     M190
      RST     M191
      RST     M1050
      RST     M1052
178   LDP     M18  ; Touch   Position Move
      ANI     L2006  ; Ax.6  Start accept flag
      ANI     L2007  ; Ax.7  Start accept flag
      AND     M20  ; Z1,Z2   POS     SAFERTY
      AND     M58  ; All home completed
      AND     M21  ; Lamp XY block   select
      SET     L8  ; ABS XY  START
186   LD      L8  ; ABS XY  START
      LD      L2006  ; Ax.6  Start accept flag
      OR      L2007  ; Ax.7  Start accept flag
      ANB
      RST     L8  ; ABS XY  START
191   LDP     M135  ; Sheet ready signal
      ANI     L2005  ; Ax.5  Start accept flag
      ANI     L2006  ; Ax.6  Start accept flag
      ANI     L2007  ; Ax.7  Start accept flag
      AND     M20  ; Z1,Z2   POS     SAFERTY
      AND     M58  ; All home completed
      SET     L18
199   LD      L18
      LD      L2006  ; Ax.6  Start accept flag
      OR      L2007  ; Ax.7  Start accept flag
      OR      L2005  ; Ax.5  Start accept flag
      ANB
      RST     L18
205   LDP     M18  ; Touch   Position Move
      ANI     L2001  ; Ax.1  Start accept flag
      AND     M22  ; Lamp Z1 block select
      AND     M58  ; All home completed
      SET     L101  ; Axis 1  (Z1)    START   ABS
211   LD      L101  ; Axis 1  (Z1)    START   ABS
      AND     L2001  ; Ax.1  Start accept flag
      RST     L101  ; Axis 1  (Z1)    START   ABS
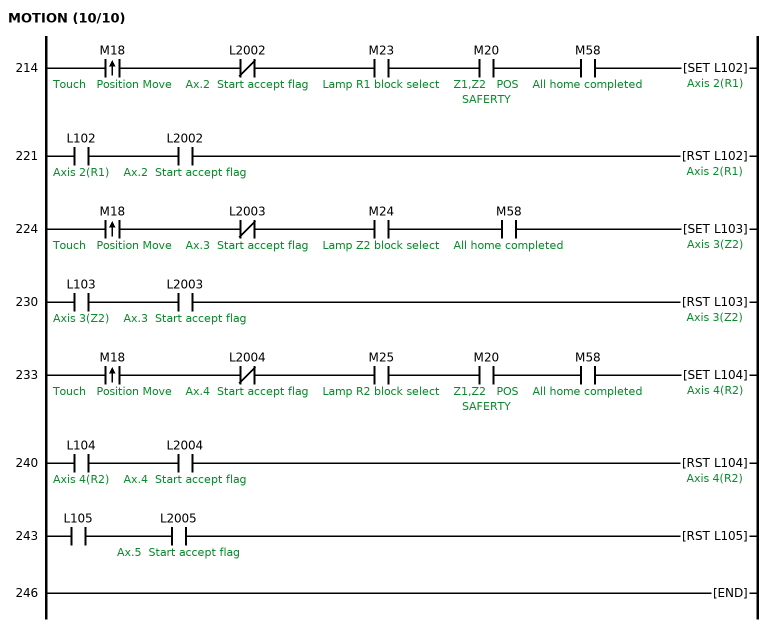
214   LDP     M18  ; Touch   Position Move
      ANI     L2002  ; Ax.2  Start accept flag
      AND     M23  ; Lamp R1 block select
      AND     M20  ; Z1,Z2   POS     SAFERTY
      AND     M58  ; All home completed
      SET     L102  ; Axis 2(R1)
221   LD      L102  ; Axis 2(R1)
      AND     L2002  ; Ax.2  Start accept flag
      RST     L102  ; Axis 2(R1)
224   LDP     M18  ; Touch   Position Move
      ANI     L2003  ; Ax.3  Start accept flag
      AND     M24  ; Lamp Z2 block select
      AND     M58  ; All home completed
      SET     L103  ; Axis 3(Z2)
230   LD      L103  ; Axis 3(Z2)
      AND     L2003  ; Ax.3  Start accept flag
      RST     L103  ; Axis 3(Z2)
233   LDP     M18  ; Touch   Position Move
      ANI     L2004  ; Ax.4  Start accept flag
      AND     M25  ; Lamp R2 block select
      AND     M20  ; Z1,Z2   POS     SAFERTY
      AND     M58  ; All home completed
      SET     L104  ; Axis 4(R2)
240   LD      L104  ; Axis 4(R2)
      AND     L2004  ; Ax.4  Start accept flag
      RST     L104  ; Axis 4(R2)
243   LD      L105
      AND     L2005  ; Ax.5  Start accept flag
      RST     L105
246   END
END_PROGRAM

PROGRAM TOUCH
